{attribute 'GeneratedUsingTerminal: EL2535-0103-0023'}
{attribute addProperty BoxType "EL2535-0103-0023"}
{attribute addProperty Id "Ready_to_enableBOOL1WarningBOOL1ErrorBOOL1TxPDO_ToggleBOOL1"}
{attribute addProperty CRC "1925348992"}
{attribute addProperty Size "4"}
TYPE Status_72C27E80 :
STRUCT
	{attribute addProperty Name "Ready_to_enable"}
	Ready_to_enable : BOOL;
	{attribute addProperty Name "Warning"}
	Warning : BOOL;
	{attribute addProperty Name "Error"}
	Error : BOOL;
	{attribute addProperty Name "TxPDO_Toggle"}
	TxPDO_Toggle : BOOL;
END_STRUCT
END_TYPE

(* stored: Version 1.2.0.0, ProductVersion 3.1.4024.9
   DUT Status_72C27E80: Id {e432766f-2c3f-4df5-9d9a-4664ef89334c} *)
